# EPICS StreamDevice protocol: thorlabs/pm100usb/device_config/pm100usb.proto
Terminator = LF;

ReplyTimeout = 200;
##=====================================
##=============== Debug ===============
debug {
    out "%s";
    in "%39c";
}
##=====================================
##=============== DeviceID ============
idn {
    out "*IDN?";
    in "%#s";
}

##=====================================
##=============== Wavelength ==========
get_wavelength {
    out "SENS:CORR:WAV?";
    in "%f";
}

set_wavelength {
    out "SENS:CORR:WAV %f";
}

##=====================================
##=============== Power ===============
get_power {
    out "MEAS:POW?";
    in "%f";
}

get_power_unit {
    out "SENS:POW:UNIT?";
    in "%{W|dBm}";
}

##=====================================
##=============== Current =============
get_curr {
    out "MEAS:CURR?";
    in "%f";
}

##=====================================
##=============== Voltage =============
get_volt {
    out "MEAS:VOLT?";
    in "%f";
}

##=====================================
##=============== Power Density =======
get_pdens {
    out "MEAS:PDEN?";
    in "%f";
}

##=====================================
##=============== Zeroing =============
get_zero_state {
    out "SENS:CORR:COLL:ZERO:STAT?";
    in "%i";
}

set_zero {
    out "SENS:CORR:COLL:ZERO:INIT";
    @init{
        get_zero_state;
    }
}

##=====================================
##=============== Zeroing =============
get_aver {
    out "SENS:AVER?";
    in "%d";
    @init{
        out "SENS:AVER?";
        in "%d";
    }
}

set_aver {
    out "SENS:AVER %d";
    @init{
        get_aver;
    }
}
